ABB RobotStudio station: NLP2Commands_IRB140.rspag

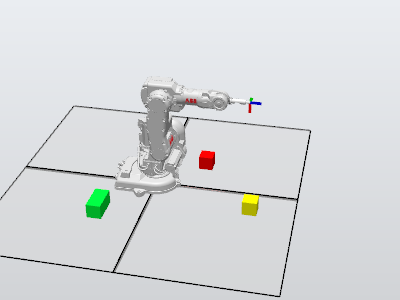
--- station ---
Station FinalProject (saved by RobotStudio 24.4.11080.0)
Controller IRB140_6_81
  mechanical unit ROB_1: IRB140_6_81, 6 joints, base frame (0, 0, 0) mm
Layout (positions relative to the parent item):
  - IRB140_6_81 [mechanism, from %ABB.RobotStudio.Models.IRB140%\IRB140_6_81_C_G_03.rslib] at (0, 0, 0) mm; joint values [0, 0, 0, 0, 0, 0] (rad or m)
  - VacuumGripper [mechanism] at (515, 0, 712) mm, rotated rx 0 ry 90 rz 0 deg
      TCP VacuumGripper at (122.78, 0, 0) mm, rotated rx 90 ry 45 rz 90 deg
      links: FakeEE
  - Cubo rojo [part] at (9, 9, 0) mm, size 100 x 100 x 100 mm
  - Cubo amarillo [part] at (0, 0, 0) mm, size 100 x 100 x 100 mm
  - Rectángulo verde [part] at (0, 0, 0) mm, size 100 x 200 x 100 mm
  - Cubo rojo [smart component, from Components\Positioner.rslib]
      properties: Object=Cubo rojo; Position=[0.009 0.009 0]; Orientation=[0 0 0]; Reference=Global; ReferenceObject=(none)
  - Cubo amarillo [smart component, from Components\Positioner.rslib]
      properties: Object=Cubo amarillo; Position=[0 0 0]; Orientation=[0 0 0]; Reference=Global; ReferenceObject=(none)
  - Rectángulo verde [smart component, from Components\Positioner.rslib]
      properties: Object=Rectángulo verde; Position=[0 0 0]; Orientation=[0 0 0]; Reference=Global; ReferenceObject=(none)
  - Detacher [smart component, from Components\Detacher.rslib]
      properties: Child=Cubo rojo; KeepPosition=true
  - Detacher_2 [smart component, from Components\Detacher.rslib]
      properties: Child=Cubo amarillo; KeepPosition=true
  - Detacher_3 [smart component, from Components\Detacher.rslib]
      properties: Child=Rectángulo verde; KeepPosition=true
  - Attacher [smart component, from Components\Attacher.rslib]
      properties: Parent=VacuumGripper; Flange=0; Child=Cubo rojo; Mount=false; Offset=[0 0 0]; Orientation=[0 0 0]
  - Attacher_2 [smart component, from Components\Attacher.rslib]
      properties: Parent=VacuumGripper; Flange=0; Child=Cubo amarillo; Mount=false; Offset=[0 0 0]; Orientation=[0 0 0]
  - Attacher_3 [smart component, from Components\Attacher.rslib]
      properties: Parent=VacuumGripper; Flange=0; Child=Rectángulo verde; Mount=false; Offset=[0 0 0]; Orientation=[0 0 0]
  - PlaneSensor [smart component, from Components\PlaneSensor.rslib]
      properties: Origin=[0.25 0.25 0.101]; Axis1=[0.1 0 0]; Axis2=[0 0.1 0]; Tag=(none); SensedPart=(none)
    - _sensorPart_ [part], size 100 x 100 x 0 mm
  - PlaneSensor_2 [smart component, from Components\PlaneSensor.rslib]
      properties: Origin=[0.65 -0.25 0.101]; Axis1=[0.1 0 0]; Axis2=[0 0.1 0]; Tag=(none); SensedPart=Cubo amarillo
    - _sensorPart_ [part], size 100 x 100 x 0 mm
  - PlaneSensor_3 [smart component, from Components\PlaneSensor.rslib]
      properties: Origin=[-0.35 -0.5 0.101]; Axis1=[0.1 0 0]; Axis2=[0 0.2 0]; Tag=(none); SensedPart=(none)
    - _sensorPart_ [part], size 100 x 200 x 0 mm
Attachment: VacuumGripper is attached to IRB140_6_81 / Link6
Station signals: DI Reset_posiciones
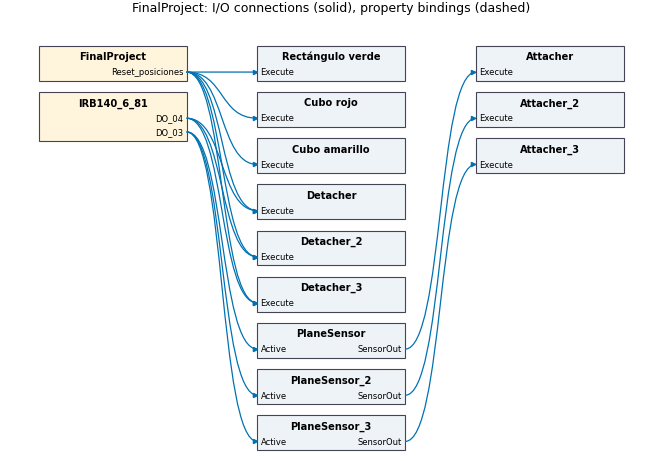
Station logic (signal -> signal, property => property):
  FinalProject.Reset_posiciones -> Rectángulo verde.Execute
  FinalProject.Reset_posiciones -> Cubo rojo.Execute
  FinalProject.Reset_posiciones -> Cubo amarillo.Execute
  IRB140_6_81.DO_04 -> Detacher.Execute
  IRB140_6_81.DO_04 -> Detacher_2.Execute
  IRB140_6_81.DO_04 -> Detacher_3.Execute
  FinalProject.Reset_posiciones -> Detacher.Execute
  FinalProject.Reset_posiciones -> Detacher_2.Execute
  FinalProject.Reset_posiciones -> Detacher_3.Execute
  PlaneSensor.SensorOut -> Attacher.Execute
  PlaneSensor_2.SensorOut -> Attacher_2.Execute
  PlaneSensor_3.SensorOut -> Attacher_3.Execute
  IRB140_6_81.DO_03 -> PlaneSensor.Active
  IRB140_6_81.DO_03 -> PlaneSensor_2.Active
  IRB140_6_81.DO_03 -> PlaneSensor_3.Active
Targets, tools, work objects and paths stored in the station and not in the controller backup, written as RAPID:
! task T_ROB1
MODULE Numbers
  CONST robtarget T_01:=[[-310.742,318.894,0],[1,0,0,0],[0,0,0,0],[9E+09,9E+09,9E+09,9E+09,9E+09,9E+09]];
  CONST robtarget T_02:=[[-285.702,367.273,0],[1,0,0,0],[0,-1,0,0],[9E+09,9E+09,9E+09,9E+09,9E+09,9E+09]];
  CONST robtarget T_03:=[[-206.529,382.913,0],[1,0,0,0],[0,-1,0,0],[9E+09,9E+09,9E+09,9E+09,9E+09,9E+09]];
  CONST robtarget T_04:=[[-128.165,367.435,0],[1,0,0,0],[0,-2,1,0],[9E+09,9E+09,9E+09,9E+09,9E+09,9E+09]];
  CONST robtarget T_05:=[[-102.477,318.894,0],[1,0,0,0],[-2,0,1,6],[9E+09,9E+09,9E+09,9E+09,9E+09,9E+09]];
  CONST robtarget T_06:=[[-127.679,270.676,0],[1,0,0,0],[-2,0,1,6],[9E+09,9E+09,9E+09,9E+09,9E+09,9E+09]];
  CONST robtarget T_07:=[[-206.691,255.036,0],[1,0,0,0],[-1,0,-1,0],[9E+09,9E+09,9E+09,9E+09,9E+09,9E+09]];
  CONST robtarget T_08:=[[-284.811,270.514,0],[1,0,0,0],[-1,0,-1,0],[9E+09,9E+09,9E+09,9E+09,9E+09,9E+09]];
  CONST robtarget T_09:=[[-310.742,318.894,0],[1,0,0,0],[0,-1,0,0],[9E+09,9E+09,9E+09,9E+09,9E+09,9E+09]];
  CONST robtarget T_11:=[[-106.691,366.707,0],[1,0,0,0],[0,0,-1,1],[9E+09,9E+09,9E+09,9E+09,9E+09,9E+09]];
  CONST robtarget T_12:=[[-106.691,269.138,0],[1,0,0,0],[0,0,-1,1],[9E+09,9E+09,9E+09,9E+09,9E+09,9E+09]];
  CONST robtarget T_13:=[[-106.691,317.923,0],[1,0,0,0],[0,0,-1,1],[9E+09,9E+09,9E+09,9E+09,9E+09,9E+09]];
  CONST robtarget T_14:=[[-307.339,315.005,0],[1,0,0,0],[0,0,-1,1],[9E+09,9E+09,9E+09,9E+09,9E+09,9E+09]];
  CONST robtarget T_15:=[[-285.297,336.399,0],[1,0,0,0],[0,1,-2,1],[9E+09,9E+09,9E+09,9E+09,9E+09,9E+09]];
  CONST robtarget T_16:=[[-279.462,366.707,0],[1,0,0,0],[0,1,-2,1],[9E+09,9E+09,9E+09,9E+09,9E+09,9E+09]];
  CONST robtarget T_21:=[[-106.691,261.009,0],[1,0,0,0],[0,-1,0,0],[9E+09,9E+09,9E+09,9E+09,9E+09,9E+09]];
  CONST robtarget T_22:=[[-106.691,384.347,0],[1,0,0,0],[0,-2,1,0],[9E+09,9E+09,9E+09,9E+09,9E+09,9E+09]];
  CONST robtarget T_23:=[[-129.867,359.226,0],[1,0,0,0],[0,-2,1,0],[9E+09,9E+09,9E+09,9E+09,9E+09,9E+09]];
  CONST robtarget T_24:=[[-153.206,334.509,0],[1,0,0,0],[0,-2,1,0],[9E+09,9E+09,9E+09,9E+09,9E+09,9E+09]];
  CONST robtarget T_25:=[[-181.731,306.39,0],[1,0,0,0],[0,-1,0,0],[9E+09,9E+09,9E+09,9E+09,9E+09,9E+09]];
  CONST robtarget T_26:=[[-215.929,279.647,0],[1,0,0,0],[0,-1,0,0],[9E+09,9E+09,9E+09,9E+09,9E+09,9E+09]];
  CONST robtarget T_27:=[[-255.961,269.274,0],[1,0,0,0],[0,-1,0,0],[9E+09,9E+09,9E+09,9E+09,9E+09,9E+09]];
  CONST robtarget T_28:=[[-296.075,285.077,0],[1,0,0,0],[0,-1,0,0],[9E+09,9E+09,9E+09,9E+09,9E+09,9E+09]];
  CONST robtarget T_29:=[[-310.905,328.918,0],[1,0,0,0],[0,-1,0,0],[9E+09,9E+09,9E+09,9E+09,9E+09,9E+09]];
  CONST robtarget T_210:=[[-306.934,357.038,0],[1,0,0,0],[0,-1,0,0],[9E+09,9E+09,9E+09,9E+09,9E+09,9E+09]];
  CONST robtarget T_211:=[[-298.911,380.133,0],[1,0,0,0],[0,-1,0,0],[9E+09,9E+09,9E+09,9E+09,9E+09,9E+09]];
  CONST robtarget T_31:=[[-298.587,375.377,0],[1,0,0,0],[0,-1,0,0],[9E+09,9E+09,9E+09,9E+09,9E+09,9E+09]];
  CONST robtarget T_32:=[[-307.096,351.633,0],[1,0,0,0],[0,-1,0,0],[9E+09,9E+09,9E+09,9E+09,9E+09,9E+09]];
  CONST robtarget T_33:=[[-310.905,323.189,0],[1,0,0,0],[0,-1,0,0],[9E+09,9E+09,9E+09,9E+09,9E+09,9E+09]];
  CONST robtarget T_34:=[[-308.149,299.445,0],[1,0,0,0],[0,-1,0,0],[9E+09,9E+09,9E+09,9E+09,9E+09,9E+09]];
  CONST robtarget T_35:=[[-299.559,281.049,0],[1,0,0,0],[0,-1,0,0],[9E+09,9E+09,9E+09,9E+09,9E+09,9E+09]];
  CONST robtarget T_36:=[[-284.081,267.759,0],[1,0,0,0],[0,-1,0,0],[9E+09,9E+09,9E+09,9E+09,9E+09,9E+09]];
  CONST robtarget T_37:=[[-262.606,263.221,0],[1,0,0,0],[0,-1,0,0],[9E+09,9E+09,9E+09,9E+09,9E+09,9E+09]];
  CONST robtarget T_38:=[[-233.595,274.08,0],[1,0,0,0],[0,-1,0,0],[9E+09,9E+09,9E+09,9E+09,9E+09,9E+09]];
  CONST robtarget T_39:=[[-217.874,300.174,0],[1,0,0,0],[0,-1,0,0],[9E+09,9E+09,9E+09,9E+09,9E+09,9E+09]];
  CONST robtarget T_310:=[[-215.199,340.044,0],[1,0,0,0],[0,-1,0,0],[9E+09,9E+09,9E+09,9E+09,9E+09,9E+09]];
  CONST robtarget T_311:=[[-215.929,300.174,0],[1,0,0,0],[0,-1,0,0],[9E+09,9E+09,9E+09,9E+09,9E+09,9E+09]];
  CONST robtarget T_312:=[[-202.963,273.27,0],[1,0,0,0],[0,-1,0,0],[9E+09,9E+09,9E+09,9E+09,9E+09,9E+09]];
  CONST robtarget T_313:=[[-188.214,263.221,0],[1,0,0,0],[0,-1,0,0],[9E+09,9E+09,9E+09,9E+09,9E+09,9E+09]];
  CONST robtarget T_314:=[[-166.01,259.331,0],[1,0,0,0],[0,-1,0,0],[9E+09,9E+09,9E+09,9E+09,9E+09,9E+09]];
  CONST robtarget T_315:=[[-141.131,263.95,0],[1,0,0,0],[0,-1,0,0],[9E+09,9E+09,9E+09,9E+09,9E+09,9E+09]];
  CONST robtarget T_316:=[[-120.953,276.997,0],[1,0,0,0],[0,-1,0,0],[9E+09,9E+09,9E+09,9E+09,9E+09,9E+09]];
  CONST robtarget T_317:=[[-107.177,298.148,0],[1,0,0,0],[0,-2,1,0],[9E+09,9E+09,9E+09,9E+09,9E+09,9E+09]];
  CONST robtarget T_318:=[[-102.477,326.268,0],[1,0,0,0],[0,-2,1,0],[9E+09,9E+09,9E+09,9E+09,9E+09,9E+09]];
  CONST robtarget T_319:=[[-106.123,356.09,0],[1,0,0,0],[0,-2,1,0],[9E+09,9E+09,9E+09,9E+09,9E+09,9E+09]];
  CONST robtarget T_320:=[[-114.794,380.887,0],[1,0,0,0],[0,-2,1,0],[9E+09,9E+09,9E+09,9E+09,9E+09,9E+09]];
  CONST robtarget T_41:=[[-106.691,281.323,0],[1,0,0,0],[-1,-1,0,1],[9E+09,9E+09,9E+09,9E+09,9E+09,9E+09]];
  CONST robtarget T_42:=[[-306.691,281.323,0],[1,0,0,0],[0,0,-1,1],[9E+09,9E+09,9E+09,9E+09,9E+09,9E+09]];
  CONST robtarget T_43:=[[-306.691,305.958,0],[1,0,0,0],[0,1,-2,1],[9E+09,9E+09,9E+09,9E+09,9E+09,9E+09]];
  CONST robtarget T_44:=[[-203.611,395.424,0],[1,0,0,0],[0,1,-2,1],[9E+09,9E+09,9E+09,9E+09,9E+09,9E+09]];
  CONST robtarget T_45:=[[-175.41,395.424,0],[1,0,0,0],[0,1,-2,1],[9E+09,9E+09,9E+09,9E+09,9E+09,9E+09]];
  CONST robtarget T_46:=[[-175.41,257.498,0],[1,0,0,0],[0,1,-2,1],[9E+09,9E+09,9E+09,9E+09,9E+09,9E+09]];
  CONST robtarget T_51:=[[-306.691,269.007,0],[1,0,0,0],[0,1,-2,1],[9E+09,9E+09,9E+09,9E+09,9E+09,9E+09]];
  CONST robtarget T_52:=[[-306.691,378.732,0],[1,0,0,0],[0,1,-2,1],[9E+09,9E+09,9E+09,9E+09,9E+09,9E+09]];
  CONST robtarget T_53:=[[-223.611,378.732,0],[1,0,0,0],[0,1,-2,1],[9E+09,9E+09,9E+09,9E+09,9E+09,9E+09]];
  CONST robtarget T_54:=[[-229.867,352.962,0],[1,0,0,0],[0,1,-2,1],[9E+09,9E+09,9E+09,9E+09,9E+09,9E+09]];
  CONST robtarget T_55:=[[-231.002,334.809,0],[1,0,0,0],[0,1,-2,1],[9E+09,9E+09,9E+09,9E+09,9E+09,9E+09]];
  CONST robtarget T_56:=[[-228.49,308.796,0],[1,0,0,0],[0,1,-2,1],[9E+09,9E+09,9E+09,9E+09,9E+09,9E+09]];
  CONST robtarget T_57:=[[-218.522,288.456,0],[1,0,0,0],[0,1,-2,1],[9E+09,9E+09,9E+09,9E+09,9E+09,9E+09]];
  CONST robtarget T_58:=[[-199.721,273.221,0],[1,0,0,0],[0,1,-2,1],[9E+09,9E+09,9E+09,9E+09,9E+09,9E+09]];
  CONST robtarget T_59:=[[-170.224,267.873,0],[1,0,0,0],[0,1,-2,1],[9E+09,9E+09,9E+09,9E+09,9E+09,9E+09]];
  CONST robtarget T_510:=[[-143.482,272.492,0],[1,0,0,0],[0,0,-1,1],[9E+09,9E+09,9E+09,9E+09,9E+09,9E+09]];
  CONST robtarget T_511:=[[-122.088,285.539,0],[1,0,0,0],[0,0,-1,1],[9E+09,9E+09,9E+09,9E+09,9E+09,9E+09]];
  CONST robtarget T_512:=[[-107.744,306.527,0],[1,0,0,0],[0,0,-1,1],[9E+09,9E+09,9E+09,9E+09,9E+09,9E+09]];
  CONST robtarget T_513:=[[-102.477,334.647,0],[1,0,0,0],[0,0,-1,1],[9E+09,9E+09,9E+09,9E+09,9E+09,9E+09]];
  CONST robtarget T_514:=[[-105.637,362.848,0],[1,0,0,0],[0,0,-1,1],[9E+09,9E+09,9E+09,9E+09,9E+09,9E+09]];
  CONST robtarget T_515:=[[-113.822,386.997,0],[1,0,0,0],[0,0,-1,1],[9E+09,9E+09,9E+09,9E+09,9E+09,9E+09]];
  CONST robtarget T_61:=[[-307.663,280.947,0],[1,0,0,0],[0,0,-1,1],[9E+09,9E+09,9E+09,9E+09,9E+09,9E+09]];
  CONST robtarget T_62:=[[-310.418,303.638,0],[1,0,0,0],[0,1,-2,1],[9E+09,9E+09,9E+09,9E+09,9E+09,9E+09]];
  CONST robtarget T_63:=[[-301.909,343.346,0],[1,0,0,0],[0,1,-2,1],[9E+09,9E+09,9E+09,9E+09,9E+09,9E+09]];
  CONST robtarget T_64:=[[-278.165,371.385,0],[1,0,0,0],[0,1,-2,1],[9E+09,9E+09,9E+09,9E+09,9E+09,9E+09]];
  CONST robtarget T_65:=[[-241.618,387.916,0],[1,0,0,0],[0,1,-2,1],[9E+09,9E+09,9E+09,9E+09,9E+09,9E+09]];
  CONST robtarget T_66:=[[-194.535,393.265,0],[1,0,0,0],[0,1,-2,1],[9E+09,9E+09,9E+09,9E+09,9E+09,9E+09]];
  CONST robtarget T_67:=[[-149.721,387.43,0],[1,0,0,0],[0,1,-2,1],[9E+09,9E+09,9E+09,9E+09,9E+09,9E+09]];
  CONST robtarget T_68:=[[-120.629,371.223,0],[1,0,0,0],[0,0,-1,1],[9E+09,9E+09,9E+09,9E+09,9E+09,9E+09]];
  CONST robtarget T_69:=[[-107.015,351.693,0],[1,0,0,0],[0,0,-1,1],[9E+09,9E+09,9E+09,9E+09,9E+09,9E+09]];
  CONST robtarget T_610:=[[-102.477,327.138,0],[1,0,0,0],[0,0,-1,1],[9E+09,9E+09,9E+09,9E+09,9E+09,9E+09]];
  CONST robtarget T_611:=[[-107.258,302.503,0],[1,0,0,0],[0,0,-1,1],[9E+09,9E+09,9E+09,9E+09,9E+09,9E+09]];
  CONST robtarget T_612:=[[-121.277,282.406,0],[1,0,0,0],[0,0,-1,1],[9E+09,9E+09,9E+09,9E+09,9E+09,9E+09]];
  CONST robtarget T_613:=[[-143.076,268.71,0],[1,0,0,0],[0,0,-1,1],[9E+09,9E+09,9E+09,9E+09,9E+09,9E+09]];
  CONST robtarget T_614:=[[-171.52,263.605,0],[1,0,0,0],[0,1,-2,1],[9E+09,9E+09,9E+09,9E+09,9E+09,9E+09]];
  CONST robtarget T_615:=[[-201.504,268.954,0],[1,0,0,0],[0,1,-2,1],[9E+09,9E+09,9E+09,9E+09,9E+09,9E+09]];
  CONST robtarget T_616:=[[-222.574,285.323,0],[1,0,0,0],[0,1,-2,1],[9E+09,9E+09,9E+09,9E+09,9E+09,9E+09]];
  CONST robtarget T_617:=[[-232.055,303.638,0],[1,0,0,0],[0,1,-2,1],[9E+09,9E+09,9E+09,9E+09,9E+09,9E+09]];
  CONST robtarget T_618:=[[-234.405,324.059,0],[1,0,0,0],[0,1,-2,1],[9E+09,9E+09,9E+09,9E+09,9E+09,9E+09]];
  CONST robtarget T_619:=[[-230.759,346.101,0],[1,0,0,0],[0,1,-2,1],[9E+09,9E+09,9E+09,9E+09,9E+09,9E+09]];
  CONST robtarget T_620:=[[-220.467,365.712,0],[1,0,0,0],[0,1,-2,1],[9E+09,9E+09,9E+09,9E+09,9E+09,9E+09]];
  CONST robtarget T_621:=[[-194.535,393.265,0],[1,0,0,0],[0,1,-2,1],[9E+09,9E+09,9E+09,9E+09,9E+09,9E+09]];
  CONST robtarget T_71:=[[-306.691,388.239,0],[1,0,0,0],[0,-1,0,0],[9E+09,9E+09,9E+09,9E+09,9E+09,9E+09]];
  CONST robtarget T_72:=[[-306.691,261.334,0],[1,0,0,0],[0,-1,0,0],[9E+09,9E+09,9E+09,9E+09,9E+09,9E+09]];
  CONST robtarget T_73:=[[-106.691,347.882,0],[1,0,0,0],[0,-1,0,0],[9E+09,9E+09,9E+09,9E+09,9E+09,9E+09]];
  CONST robtarget T_81:=[[-214.308,359.688,0],[1,0,0,0],[0,1,-2,1],[9E+09,9E+09,9E+09,9E+09,9E+09,9E+09]];
  CONST robtarget T_82:=[[-233.109,381.568,0],[1,0,0,0],[0,1,-2,1],[9E+09,9E+09,9E+09,9E+09,9E+09,9E+09]];
  CONST robtarget T_83:=[[-258.554,388.699,0],[1,0,0,0],[0,1,-2,1],[9E+09,9E+09,9E+09,9E+09,9E+09,9E+09]];
  CONST robtarget T_84:=[[-296.156,371.681,0],[1,0,0,0],[0,1,-2,1],[9E+09,9E+09,9E+09,9E+09,9E+09,9E+09]];
  CONST robtarget T_85:=[[-311.229,328.407,0],[1,0,0,0],[0,1,-2,1],[9E+09,9E+09,9E+09,9E+09,9E+09,9E+09]];
  CONST robtarget T_86:=[[-296.966,284.728,0],[1,0,0,0],[0,1,-2,1],[9E+09,9E+09,9E+09,9E+09,9E+09,9E+09]];
  CONST robtarget T_87:=[[-260.337,268.278,0],[1,0,0,0],[0,1,-2,1],[9E+09,9E+09,9E+09,9E+09,9E+09,9E+09]];
  CONST robtarget T_88:=[[-233.757,276.138,0],[1,0,0,0],[0,1,-2,1],[9E+09,9E+09,9E+09,9E+09,9E+09,9E+09]];
  CONST robtarget T_89:=[[-213.174,298.748,0],[1,0,0,0],[0,1,-2,1],[9E+09,9E+09,9E+09,9E+09,9E+09,9E+09]];
  CONST robtarget T_810:=[[-213.498,359.688,0],[1,0,0,0],[0,1,-2,1],[9E+09,9E+09,9E+09,9E+09,9E+09,9E+09]];
  CONST robtarget T_811:=[[-191.78,384.89,0],[1,0,0,0],[0,1,-2,1],[9E+09,9E+09,9E+09,9E+09,9E+09,9E+09]];
  CONST robtarget T_812:=[[-161.958,393.561,0],[1,0,0,0],[0,1,-2,1],[9E+09,9E+09,9E+09,9E+09,9E+09,9E+09]];
  CONST robtarget T_813:=[[-138.457,389.185,0],[1,0,0,0],[0,0,-1,1],[9E+09,9E+09,9E+09,9E+09,9E+09,9E+09]];
  CONST robtarget T_814:=[[-119.332,376.381,0],[1,0,0,0],[0,0,-1,1],[9E+09,9E+09,9E+09,9E+09,9E+09,9E+09]];
  CONST robtarget T_815:=[[-106.61,355.555,0],[1,0,0,0],[0,0,-1,1],[9E+09,9E+09,9E+09,9E+09,9E+09,9E+09]];
  CONST robtarget T_816:=[[-102.152,328.407,0],[1,0,0,0],[0,0,-1,1],[9E+09,9E+09,9E+09,9E+09,9E+09,9E+09]];
  CONST robtarget T_817:=[[-119.494,281.892,0],[1,0,0,0],[0,0,-1,1],[9E+09,9E+09,9E+09,9E+09,9E+09,9E+09]];
  CONST robtarget T_818:=[[-162.444,263.253,0],[1,0,0,0],[0,1,-2,1],[9E+09,9E+09,9E+09,9E+09,9E+09,9E+09]];
  CONST robtarget T_819:=[[-192.59,272.249,0],[1,0,0,0],[0,1,-2,1],[9E+09,9E+09,9E+09,9E+09,9E+09,9E+09]];
  CONST robtarget T_820:=[[-212.363,298.748,0],[1,0,0,0],[0,1,-2,1],[9E+09,9E+09,9E+09,9E+09,9E+09,9E+09]];
  CONST robtarget T_821:=[[-214.308,359.688,0],[1,0,0,0],[0,1,-2,1],[9E+09,9E+09,9E+09,9E+09,9E+09,9E+09]];
  CONST robtarget T_91:=[[-105.556,371.949,0],[1,0,0,0],[0,0,-1,1],[9E+09,9E+09,9E+09,9E+09,9E+09,9E+09]];
  CONST robtarget T_92:=[[-102.801,349.258,0],[1,0,0,0],[0,0,-1,1],[9E+09,9E+09,9E+09,9E+09,9E+09,9E+09]];
  CONST robtarget T_93:=[[-110.986,309.388,0],[1,0,0,0],[0,0,-1,1],[9E+09,9E+09,9E+09,9E+09,9E+09,9E+09]];
  CONST robtarget T_94:=[[-134.729,281.673,0],[1,0,0,0],[0,0,-1,1],[9E+09,9E+09,9E+09,9E+09,9E+09,9E+09]];
  CONST robtarget T_95:=[[-171.682,265.223,0],[1,0,0,0],[0,1,-2,1],[9E+09,9E+09,9E+09,9E+09,9E+09,9E+09]];
  CONST robtarget T_96:=[[-218.684,259.631,0],[1,0,0,0],[0,1,-2,1],[9E+09,9E+09,9E+09,9E+09,9E+09,9E+09]];
  CONST robtarget T_97:=[[-263.903,265.304,0],[1,0,0,0],[0,1,-2,1],[9E+09,9E+09,9E+09,9E+09,9E+09,9E+09]];
  CONST robtarget T_98:=[[-292.752,281.349,0],[1,0,0,0],[0,1,-2,1],[9E+09,9E+09,9E+09,9E+09,9E+09,9E+09]];
  CONST robtarget T_99:=[[-306.123,300.798,0],[1,0,0,0],[0,1,-2,1],[9E+09,9E+09,9E+09,9E+09,9E+09,9E+09]];
  CONST robtarget T_910:=[[-310.742,325.757,0],[1,0,0,0],[0,1,-2,1],[9E+09,9E+09,9E+09,9E+09,9E+09,9E+09]];
  CONST robtarget T_911:=[[-305.799,350.15,0],[1,0,0,0],[0,1,-2,1],[9E+09,9E+09,9E+09,9E+09,9E+09,9E+09]];
  CONST robtarget T_912:=[[-291.942,370.49,0],[1,0,0,0],[0,1,-2,1],[9E+09,9E+09,9E+09,9E+09,9E+09,9E+09]];
  CONST robtarget T_913:=[[-269.9,384.266,0],[1,0,0,0],[0,1,-2,1],[9E+09,9E+09,9E+09,9E+09,9E+09,9E+09]];
  CONST robtarget T_914:=[[-241.699,389.291,0],[1,0,0,0],[0,1,-2,1],[9E+09,9E+09,9E+09,9E+09,9E+09,9E+09]];
  CONST robtarget T_915:=[[-211.472,383.78,0],[1,0,0,0],[0,1,-2,1],[9E+09,9E+09,9E+09,9E+09,9E+09,9E+09]];
  CONST robtarget T_916:=[[-190.645,367.573,0],[1,0,0,0],[0,1,-2,1],[9E+09,9E+09,9E+09,9E+09,9E+09,9E+09]];
  CONST robtarget T_917:=[[-181.245,349.177,0],[1,0,0,0],[0,1,-2,1],[9E+09,9E+09,9E+09,9E+09,9E+09,9E+09]];
  CONST robtarget T_918:=[[-178.814,328.999,0],[1,0,0,0],[0,1,-2,1],[9E+09,9E+09,9E+09,9E+09,9E+09,9E+09]];
  CONST robtarget T_919:=[[-182.136,307.767,0],[1,0,0,0],[0,1,-2,1],[9E+09,9E+09,9E+09,9E+09,9E+09,9E+09]];
  CONST robtarget T_920:=[[-192.752,287.346,0],[1,0,0,0],[0,1,-2,1],[9E+09,9E+09,9E+09,9E+09,9E+09,9E+09]];
  CONST robtarget T_921:=[[-218.684,259.631,0],[1,0,0,0],[0,1,-2,1],[9E+09,9E+09,9E+09,9E+09,9E+09,9E+09]];
  CONST robtarget T_921_2:=[[-218.684,259.631,0],[1,0,0,0],[-1,-2,1,1],[9E+09,9E+09,9E+09,9E+09,9E+09,9E+09]];
  CONST robtarget T_01_2:=[[-310.742,318.894,0],[1,0,0,0],[0,0,0,0],[9E+09,9E+09,9E+09,9E+09,9E+09,9E+09]];
  CONST robtarget T_02_2:=[[-285.702,367.273,0],[1,0,0,0],[-1,0,-1,0],[9E+09,9E+09,9E+09,9E+09,9E+09,9E+09]];
  CONST robtarget T_03_2:=[[-206.529,382.913,0],[1,0,0,0],[-1,0,-1,0],[9E+09,9E+09,9E+09,9E+09,9E+09,9E+09]];
  CONST robtarget T_04_2:=[[-128.165,367.435,0],[1,0,0,0],[-1,0,-1,0],[9E+09,9E+09,9E+09,9E+09,9E+09,9E+09]];
  CONST robtarget T_05_2:=[[-102.477,318.894,0],[1,0,0,0],[-1,0,-1,0],[9E+09,9E+09,9E+09,9E+09,9E+09,9E+09]];
  CONST robtarget T_06_2:=[[-127.679,270.676,0],[1,0,0,0],[-1,1,-2,0],[9E+09,9E+09,9E+09,9E+09,9E+09,9E+09]];
  CONST robtarget T_07_2:=[[-206.691,255.036,0],[1,0,0,0],[-1,0,-1,0],[9E+09,9E+09,9E+09,9E+09,9E+09,9E+09]];
  CONST robtarget T_08_2:=[[-284.811,270.514,0],[1,0,0,0],[-1,0,-1,0],[9E+09,9E+09,9E+09,9E+09,9E+09,9E+09]];
  CONST robtarget T_09_2:=[[-310.742,318.894,0],[1,0,0,0],[-1,0,-1,0],[9E+09,9E+09,9E+09,9E+09,9E+09,9E+09]];
  CONST robtarget T_11_2:=[[-106.691,366.707,0],[1,0,0,0],[-1,1,-2,0],[9E+09,9E+09,9E+09,9E+09,9E+09,9E+09]];
  CONST robtarget T_12_2:=[[-106.691,269.138,0],[1,0,0,0],[-1,1,-2,0],[9E+09,9E+09,9E+09,9E+09,9E+09,9E+09]];
  CONST robtarget T_13_2:=[[-106.691,317.923,0],[1,0,0,0],[-1,1,-2,0],[9E+09,9E+09,9E+09,9E+09,9E+09,9E+09]];
  CONST robtarget T_14_2:=[[-307.339,315.005,0],[1,0,0,0],[-1,1,-2,0],[9E+09,9E+09,9E+09,9E+09,9E+09,9E+09]];
  CONST robtarget T_15_2:=[[-285.297,336.399,0],[1,0,0,0],[-1,0,-1,0],[9E+09,9E+09,9E+09,9E+09,9E+09,9E+09]];
  CONST robtarget T_16_2:=[[-279.462,366.707,0],[1,0,0,0],[-1,0,-1,0],[9E+09,9E+09,9E+09,9E+09,9E+09,9E+09]];
  CONST robtarget T_21_2:=[[-106.691,261.009,0],[1,0,0,0],[-1,1,-2,0],[9E+09,9E+09,9E+09,9E+09,9E+09,9E+09]];
  CONST robtarget T_22_2:=[[-106.691,384.347,0],[1,0,0,0],[-1,1,-2,0],[9E+09,9E+09,9E+09,9E+09,9E+09,9E+09]];
  CONST robtarget T_23_2:=[[-129.867,359.226,0],[1,0,0,0],[-1,1,-2,0],[9E+09,9E+09,9E+09,9E+09,9E+09,9E+09]];
  CONST robtarget T_24_2:=[[-153.206,334.509,0],[1,0,0,0],[-1,0,-1,0],[9E+09,9E+09,9E+09,9E+09,9E+09,9E+09]];
  CONST robtarget T_25_2:=[[-181.731,306.39,0],[1,0,0,0],[-1,0,-1,0],[9E+09,9E+09,9E+09,9E+09,9E+09,9E+09]];
  CONST robtarget T_26_2:=[[-215.929,279.647,0],[1,0,0,0],[-1,0,-1,0],[9E+09,9E+09,9E+09,9E+09,9E+09,9E+09]];
  CONST robtarget T_27_2:=[[-255.961,269.274,0],[1,0,0,0],[-1,0,-1,0],[9E+09,9E+09,9E+09,9E+09,9E+09,9E+09]];
  CONST robtarget T_28_2:=[[-296.075,285.077,0],[1,0,0,0],[-1,0,-1,0],[9E+09,9E+09,9E+09,9E+09,9E+09,9E+09]];
  CONST robtarget T_29_2:=[[-310.905,328.918,0],[1,0,0,0],[-1,0,-1,0],[9E+09,9E+09,9E+09,9E+09,9E+09,9E+09]];
  CONST robtarget T_210_2:=[[-306.934,357.038,0],[1,0,0,0],[-1,0,-1,0],[9E+09,9E+09,9E+09,9E+09,9E+09,9E+09]];
  CONST robtarget T_211_2:=[[-298.911,380.133,0],[1,0,0,0],[-1,0,-1,0],[9E+09,9E+09,9E+09,9E+09,9E+09,9E+09]];
  CONST robtarget T_31_2:=[[-298.587,375.377,0],[1,0,0,0],[0,-1,0,0],[9E+09,9E+09,9E+09,9E+09,9E+09,9E+09]];
  CONST robtarget T_32_2:=[[-307.096,351.633,0],[1,0,0,0],[-1,0,-1,0],[9E+09,9E+09,9E+09,9E+09,9E+09,9E+09]];
  CONST robtarget T_33_2:=[[-310.905,323.189,0],[1,0,0,0],[-1,0,-1,0],[9E+09,9E+09,9E+09,9E+09,9E+09,9E+09]];
  CONST robtarget T_34_2:=[[-308.149,299.445,0],[1,0,0,0],[-1,0,-1,0],[9E+09,9E+09,9E+09,9E+09,9E+09,9E+09]];
  CONST robtarget T_35_2:=[[-299.559,281.049,0],[1,0,0,0],[-1,0,-1,0],[9E+09,9E+09,9E+09,9E+09,9E+09,9E+09]];
  CONST robtarget T_36_2:=[[-284.081,267.759,0],[1,0,0,0],[-1,0,-1,0],[9E+09,9E+09,9E+09,9E+09,9E+09,9E+09]];
  CONST robtarget T_37_2:=[[-262.606,263.221,0],[1,0,0,0],[-1,0,-1,0],[9E+09,9E+09,9E+09,9E+09,9E+09,9E+09]];
  CONST robtarget T_38_2:=[[-233.595,274.08,0],[1,0,0,0],[-1,0,-1,0],[9E+09,9E+09,9E+09,9E+09,9E+09,9E+09]];
  CONST robtarget T_39_2:=[[-217.874,300.174,0],[1,0,0,0],[-1,0,-1,0],[9E+09,9E+09,9E+09,9E+09,9E+09,9E+09]];
  CONST robtarget T_310_2:=[[-215.199,340.044,0],[1,0,0,0],[0,-1,0,0],[9E+09,9E+09,9E+09,9E+09,9E+09,9E+09]];
  CONST robtarget T_311_2:=[[-215.929,300.174,0],[1,0,0,0],[0,-1,0,0],[9E+09,9E+09,9E+09,9E+09,9E+09,9E+09]];
  CONST robtarget T_312_2:=[[-202.963,273.27,0],[1,0,0,0],[0,-1,0,0],[9E+09,9E+09,9E+09,9E+09,9E+09,9E+09]];
  CONST robtarget T_313_2:=[[-188.214,263.221,0],[1,0,0,0],[0,-1,0,0],[9E+09,9E+09,9E+09,9E+09,9E+09,9E+09]];
  CONST robtarget T_314_2:=[[-166.01,259.331,0],[1,0,0,0],[0,-1,0,0],[9E+09,9E+09,9E+09,9E+09,9E+09,9E+09]];
  CONST robtarget T_315_2:=[[-141.131,263.95,0],[1,0,0,0],[0,-1,0,0],[9E+09,9E+09,9E+09,9E+09,9E+09,9E+09]];
  CONST robtarget T_316_2:=[[-120.953,276.997,0],[1,0,0,0],[-1,1,-2,0],[9E+09,9E+09,9E+09,9E+09,9E+09,9E+09]];
  CONST robtarget T_317_2:=[[-107.177,298.148,0],[1,0,0,0],[-1,1,-2,0],[9E+09,9E+09,9E+09,9E+09,9E+09,9E+09]];
  CONST robtarget T_318_2:=[[-102.477,326.268,0],[1,0,0,0],[-1,1,-2,0],[9E+09,9E+09,9E+09,9E+09,9E+09,9E+09]];
  CONST robtarget T_319_2:=[[-106.123,356.09,0],[1,0,0,0],[-1,1,-2,0],[9E+09,9E+09,9E+09,9E+09,9E+09,9E+09]];
  CONST robtarget T_320_2:=[[-114.794,380.887,0],[1,0,0,0],[0,-2,1,0],[9E+09,9E+09,9E+09,9E+09,9E+09,9E+09]];
  CONST robtarget T_41_2:=[[-106.691,281.323,0],[1,0,0,0],[-1,1,-2,0],[9E+09,9E+09,9E+09,9E+09,9E+09,9E+09]];
  CONST robtarget T_42_2:=[[-306.691,281.323,0],[1,0,0,0],[-1,0,-1,0],[9E+09,9E+09,9E+09,9E+09,9E+09,9E+09]];
  CONST robtarget T_43_2:=[[-306.691,305.958,0],[1,0,0,0],[-1,0,-1,0],[9E+09,9E+09,9E+09,9E+09,9E+09,9E+09]];
  CONST robtarget T_44_2:=[[-203.611,395.424,0],[1,0,0,0],[0,-1,0,0],[9E+09,9E+09,9E+09,9E+09,9E+09,9E+09]];
  CONST robtarget T_45_2:=[[-175.41,395.424,0],[1,0,0,0],[0,-1,0,0],[9E+09,9E+09,9E+09,9E+09,9E+09,9E+09]];
  CONST robtarget T_46_2:=[[-175.41,257.498,0],[1,0,0,0],[-1,0,-1,0],[9E+09,9E+09,9E+09,9E+09,9E+09,9E+09]];
  CONST robtarget T_51_2:=[[-306.691,269.007,0],[1,0,0,0],[-1,0,-1,0],[9E+09,9E+09,9E+09,9E+09,9E+09,9E+09]];
  CONST robtarget T_52_2:=[[-306.691,378.732,0],[1,0,0,0],[0,-1,0,0],[9E+09,9E+09,9E+09,9E+09,9E+09,9E+09]];
  CONST robtarget T_53_2:=[[-223.611,378.732,0],[1,0,0,0],[0,-1,0,0],[9E+09,9E+09,9E+09,9E+09,9E+09,9E+09]];
  CONST robtarget T_54_2:=[[-229.867,352.962,0],[1,0,0,0],[-1,0,-1,0],[9E+09,9E+09,9E+09,9E+09,9E+09,9E+09]];
  CONST robtarget T_55_2:=[[-231.002,334.809,0],[1,0,0,0],[-1,0,-1,0],[9E+09,9E+09,9E+09,9E+09,9E+09,9E+09]];
  CONST robtarget T_56_2:=[[-228.49,308.796,0],[1,0,0,0],[-1,0,-1,0],[9E+09,9E+09,9E+09,9E+09,9E+09,9E+09]];
  CONST robtarget T_57_2:=[[-218.522,288.456,0],[1,0,0,0],[-1,0,-1,0],[9E+09,9E+09,9E+09,9E+09,9E+09,9E+09]];
  CONST robtarget T_58_2:=[[-199.721,273.221,0],[1,0,0,0],[-1,0,-1,0],[9E+09,9E+09,9E+09,9E+09,9E+09,9E+09]];
  CONST robtarget T_59_2:=[[-170.224,267.873,0],[1,0,0,0],[-1,0,-1,0],[9E+09,9E+09,9E+09,9E+09,9E+09,9E+09]];
  CONST robtarget T_510_2:=[[-143.482,272.492,0],[1,0,0,0],[-1,0,-1,0],[9E+09,9E+09,9E+09,9E+09,9E+09,9E+09]];
  CONST robtarget T_511_2:=[[-122.088,285.539,0],[1,0,0,0],[0,0,-1,1],[9E+09,9E+09,9E+09,9E+09,9E+09,9E+09]];
  CONST robtarget T_512_2:=[[-107.744,306.527,0],[1,0,0,0],[0,0,-1,1],[9E+09,9E+09,9E+09,9E+09,9E+09,9E+09]];
  CONST robtarget T_513_2:=[[-102.477,334.647,0],[1,0,0,0],[0,0,-1,1],[9E+09,9E+09,9E+09,9E+09,9E+09,9E+09]];
  CONST robtarget T_514_2:=[[-105.637,362.848,0],[1,0,0,0],[0,0,-1,1],[9E+09,9E+09,9E+09,9E+09,9E+09,9E+09]];
  CONST robtarget T_515_2:=[[-113.822,386.997,0],[1,0,0,0],[0,0,-1,1],[9E+09,9E+09,9E+09,9E+09,9E+09,9E+09]];
  CONST robtarget T_61_2:=[[-307.663,280.947,0],[1,0,0,0],[-1,0,-1,0],[9E+09,9E+09,9E+09,9E+09,9E+09,9E+09]];
  CONST robtarget T_62_2:=[[-310.418,303.638,0],[1,0,0,0],[-1,0,-1,0],[9E+09,9E+09,9E+09,9E+09,9E+09,9E+09]];
  CONST robtarget T_63_2:=[[-301.909,343.346,0],[1,0,0,0],[-1,0,-1,0],[9E+09,9E+09,9E+09,9E+09,9E+09,9E+09]];
  CONST robtarget T_64_2:=[[-278.165,371.385,0],[1,0,0,0],[0,-1,0,0],[9E+09,9E+09,9E+09,9E+09,9E+09,9E+09]];
  CONST robtarget T_65_2:=[[-241.618,387.916,0],[1,0,0,0],[0,-1,0,0],[9E+09,9E+09,9E+09,9E+09,9E+09,9E+09]];
  CONST robtarget T_66_2:=[[-194.535,393.265,0],[1,0,0,0],[0,-1,0,0],[9E+09,9E+09,9E+09,9E+09,9E+09,9E+09]];
  CONST robtarget T_67_2:=[[-149.721,387.43,0],[1,0,0,0],[0,-1,0,0],[9E+09,9E+09,9E+09,9E+09,9E+09,9E+09]];
  CONST robtarget T_68_2:=[[-120.629,371.223,0],[1,0,0,0],[0,-1,0,0],[9E+09,9E+09,9E+09,9E+09,9E+09,9E+09]];
  CONST robtarget T_69_2:=[[-107.015,351.693,0],[1,0,0,0],[-1,1,-2,0],[9E+09,9E+09,9E+09,9E+09,9E+09,9E+09]];
  CONST robtarget T_610_2:=[[-102.477,327.138,0],[1,0,0,0],[0,0,-1,1],[9E+09,9E+09,9E+09,9E+09,9E+09,9E+09]];
  CONST robtarget T_611_2:=[[-107.258,302.503,0],[1,0,0,0],[0,0,-1,1],[9E+09,9E+09,9E+09,9E+09,9E+09,9E+09]];
  CONST robtarget T_612_2:=[[-121.277,282.406,0],[1,0,0,0],[0,0,-1,1],[9E+09,9E+09,9E+09,9E+09,9E+09,9E+09]];
  CONST robtarget T_613_2:=[[-143.076,268.71,0],[1,0,0,0],[-1,-2,1,1],[9E+09,9E+09,9E+09,9E+09,9E+09,9E+09]];
  CONST robtarget T_614_2:=[[-171.52,263.605,0],[1,0,0,0],[-1,-2,1,1],[9E+09,9E+09,9E+09,9E+09,9E+09,9E+09]];
  CONST robtarget T_615_2:=[[-201.504,268.954,0],[1,0,0,0],[-1,-2,1,1],[9E+09,9E+09,9E+09,9E+09,9E+09,9E+09]];
  CONST robtarget T_616_2:=[[-222.574,285.323,0],[1,0,0,0],[-1,-2,1,1],[9E+09,9E+09,9E+09,9E+09,9E+09,9E+09]];
  CONST robtarget T_617_2:=[[-232.055,303.638,0],[1,0,0,0],[-1,-2,1,1],[9E+09,9E+09,9E+09,9E+09,9E+09,9E+09]];
  CONST robtarget T_618_2:=[[-234.405,324.059,0],[1,0,0,0],[-1,-2,1,1],[9E+09,9E+09,9E+09,9E+09,9E+09,9E+09]];
  CONST robtarget T_619_2:=[[-230.759,346.101,0],[1,0,0,0],[-1,-2,1,1],[9E+09,9E+09,9E+09,9E+09,9E+09,9E+09]];
  CONST robtarget T_620_2:=[[-220.467,365.712,0],[1,0,0,0],[0,1,-2,1],[9E+09,9E+09,9E+09,9E+09,9E+09,9E+09]];
  CONST robtarget T_621_2:=[[-194.535,393.265,0],[1,0,0,0],[0,1,-2,1],[9E+09,9E+09,9E+09,9E+09,9E+09,9E+09]];
  CONST robtarget T_71_2:=[[-306.691,388.239,0],[1,0,0,0],[0,-1,0,0],[9E+09,9E+09,9E+09,9E+09,9E+09,9E+09]];
  CONST robtarget T_72_2:=[[-306.691,261.334,0],[1,0,0,0],[-1,0,-1,0],[9E+09,9E+09,9E+09,9E+09,9E+09,9E+09]];
  CONST robtarget T_73_2:=[[-106.691,347.882,0],[1,0,0,0],[-1,1,-2,0],[9E+09,9E+09,9E+09,9E+09,9E+09,9E+09]];
  CONST robtarget T_81_2:=[[-214.308,359.688,0],[1,0,0,0],[-1,0,-1,0],[9E+09,9E+09,9E+09,9E+09,9E+09,9E+09]];
  CONST robtarget T_82_2:=[[-233.109,381.568,0],[1,0,0,0],[0,-1,0,0],[9E+09,9E+09,9E+09,9E+09,9E+09,9E+09]];
  CONST robtarget T_83_2:=[[-258.554,388.699,0],[1,0,0,0],[0,-1,0,0],[9E+09,9E+09,9E+09,9E+09,9E+09,9E+09]];
  CONST robtarget T_84_2:=[[-296.156,371.681,0],[1,0,0,0],[0,-1,0,0],[9E+09,9E+09,9E+09,9E+09,9E+09,9E+09]];
  CONST robtarget T_85_2:=[[-311.229,328.407,0],[1,0,0,0],[-1,0,-1,0],[9E+09,9E+09,9E+09,9E+09,9E+09,9E+09]];
  CONST robtarget T_86_2:=[[-296.966,284.728,0],[1,0,0,0],[-1,0,-1,0],[9E+09,9E+09,9E+09,9E+09,9E+09,9E+09]];
  CONST robtarget T_87_2:=[[-260.337,268.278,0],[1,0,0,0],[-1,0,-1,0],[9E+09,9E+09,9E+09,9E+09,9E+09,9E+09]];
  CONST robtarget T_88_2:=[[-233.757,276.138,0],[1,0,0,0],[-1,0,-1,0],[9E+09,9E+09,9E+09,9E+09,9E+09,9E+09]];
  CONST robtarget T_89_2:=[[-213.174,298.748,0],[1,0,0,0],[-1,0,-1,0],[9E+09,9E+09,9E+09,9E+09,9E+09,9E+09]];
  CONST robtarget T_810_2:=[[-213.498,359.688,0],[1,0,0,0],[0,1,-2,1],[9E+09,9E+09,9E+09,9E+09,9E+09,9E+09]];
  CONST robtarget T_811_2:=[[-191.78,384.89,0],[1,0,0,0],[0,1,-2,1],[9E+09,9E+09,9E+09,9E+09,9E+09,9E+09]];
  CONST robtarget T_812_2:=[[-161.958,393.561,0],[1,0,0,0],[0,1,-2,1],[9E+09,9E+09,9E+09,9E+09,9E+09,9E+09]];
  CONST robtarget T_813_2:=[[-138.457,389.185,0],[1,0,0,0],[0,0,-1,1],[9E+09,9E+09,9E+09,9E+09,9E+09,9E+09]];
  CONST robtarget T_814_2:=[[-119.332,376.381,0],[1,0,0,0],[0,0,-1,1],[9E+09,9E+09,9E+09,9E+09,9E+09,9E+09]];
  CONST robtarget T_815_2:=[[-106.61,355.555,0],[1,0,0,0],[0,0,-1,1],[9E+09,9E+09,9E+09,9E+09,9E+09,9E+09]];
  CONST robtarget T_816_2:=[[-102.152,328.407,0],[1,0,0,0],[0,0,-1,1],[9E+09,9E+09,9E+09,9E+09,9E+09,9E+09]];
  CONST robtarget T_817_2:=[[-119.494,281.892,0],[1,0,0,0],[0,0,-1,1],[9E+09,9E+09,9E+09,9E+09,9E+09,9E+09]];
  CONST robtarget T_818_2:=[[-162.444,263.253,0],[1,0,0,0],[-1,-2,1,1],[9E+09,9E+09,9E+09,9E+09,9E+09,9E+09]];
  CONST robtarget T_819_2:=[[-192.59,272.249,0],[1,0,0,0],[-1,-2,1,1],[9E+09,9E+09,9E+09,9E+09,9E+09,9E+09]];
  CONST robtarget T_820_2:=[[-212.363,298.748,0],[1,0,0,0],[-1,-2,1,1],[9E+09,9E+09,9E+09,9E+09,9E+09,9E+09]];
  CONST robtarget T_821_2:=[[-214.308,359.688,0],[1,0,0,0],[0,1,-2,1],[9E+09,9E+09,9E+09,9E+09,9E+09,9E+09]];
  CONST robtarget T_91_2:=[[-105.556,371.949,0],[1,0,0,0],[0,0,-1,1],[9E+09,9E+09,9E+09,9E+09,9E+09,9E+09]];
  CONST robtarget T_92_2:=[[-102.801,349.258,0],[1,0,0,0],[0,0,-1,1],[9E+09,9E+09,9E+09,9E+09,9E+09,9E+09]];
  CONST robtarget T_93_2:=[[-110.986,309.388,0],[1,0,0,0],[0,0,-1,1],[9E+09,9E+09,9E+09,9E+09,9E+09,9E+09]];
  CONST robtarget T_94_2:=[[-134.729,281.673,0],[1,0,0,0],[-1,-2,1,1],[9E+09,9E+09,9E+09,9E+09,9E+09,9E+09]];
  CONST robtarget T_95_2:=[[-171.682,265.223,0],[1,0,0,0],[-1,-2,1,1],[9E+09,9E+09,9E+09,9E+09,9E+09,9E+09]];
  CONST robtarget T_96_2:=[[-218.684,259.631,0],[1,0,0,0],[-1,-2,1,1],[9E+09,9E+09,9E+09,9E+09,9E+09,9E+09]];
  CONST robtarget T_97_2:=[[-263.903,265.304,0],[1,0,0,0],[-1,-2,1,1],[9E+09,9E+09,9E+09,9E+09,9E+09,9E+09]];
  CONST robtarget T_98_2:=[[-292.752,281.349,0],[1,0,0,0],[-1,-2,1,1],[9E+09,9E+09,9E+09,9E+09,9E+09,9E+09]];
  CONST robtarget T_99_2:=[[-306.123,300.798,0],[1,0,0,0],[-1,-2,1,1],[9E+09,9E+09,9E+09,9E+09,9E+09,9E+09]];
  CONST robtarget T_910_2:=[[-310.742,325.757,0],[1,0,0,0],[-1,-2,1,1],[9E+09,9E+09,9E+09,9E+09,9E+09,9E+09]];
  CONST robtarget T_911_2:=[[-305.799,350.15,0],[1,0,0,0],[0,1,-2,1],[9E+09,9E+09,9E+09,9E+09,9E+09,9E+09]];
  CONST robtarget T_912_2:=[[-291.942,370.49,0],[1,0,0,0],[0,1,-2,1],[9E+09,9E+09,9E+09,9E+09,9E+09,9E+09]];
  CONST robtarget T_913_2:=[[-269.9,384.266,0],[1,0,0,0],[0,1,-2,1],[9E+09,9E+09,9E+09,9E+09,9E+09,9E+09]];
  CONST robtarget T_914_2:=[[-241.699,389.291,0],[1,0,0,0],[0,1,-2,1],[9E+09,9E+09,9E+09,9E+09,9E+09,9E+09]];
  CONST robtarget T_915_2:=[[-211.472,383.78,0],[1,0,0,0],[0,1,-2,1],[9E+09,9E+09,9E+09,9E+09,9E+09,9E+09]];
  CONST robtarget T_916_2:=[[-190.645,367.573,0],[1,0,0,0],[0,1,-2,1],[9E+09,9E+09,9E+09,9E+09,9E+09,9E+09]];
  CONST robtarget T_917_2:=[[-181.245,349.177,0],[1,0,0,0],[-1,-2,1,1],[9E+09,9E+09,9E+09,9E+09,9E+09,9E+09]];
  CONST robtarget T_918_2:=[[-178.814,328.999,0],[1,0,0,0],[-1,-2,1,1],[9E+09,9E+09,9E+09,9E+09,9E+09,9E+09]];
  CONST robtarget T_919_2:=[[-182.136,307.767,0],[1,0,0,0],[-1,-2,1,1],[9E+09,9E+09,9E+09,9E+09,9E+09,9E+09]];
  CONST robtarget T_920_2:=[[-192.752,287.346,0],[1,0,0,0],[-1,-2,1,1],[9E+09,9E+09,9E+09,9E+09,9E+09,9E+09]];
  TASK PERS wobjdata Board:=[FALSE,TRUE,"",[[350,-300,450],[0,0,1,0]],[[0,0,0],[1,0,0,0]]];
ENDMODULE

! task T_ROB1
MODULE MainModule
  VAR robtarget goal:=[[0,0,0],[1,0,0,0],[0,0,0,0],[9E+09,9E+09,9E+09,9E+09,9E+09,9E+09]];
  VAR robtarget targetDraw:=[[0,0,0],[1,0,0,0],[0,0,0,0],[9E+09,9E+09,9E+09,9E+09,9E+09,9E+09]];
  CONST jointtarget jointHome:=[[0,0,0,0,0,0],[0,0,0,0,0,0]];
  PROC connection()
    SetDO DO_01,1;
    SetDO DO_02,0;
    SetDO DO_03,0;
  ENDPROC
  PROC disconnection()
    SetDO DO_01,0;
    SetDO DO_02,1;
    SetDO DO_03,0;
    SetDO DO_04,0;
    SetDO DO_05,1;
  ENDPROC
  PROC getOrders()
    SetDO DO_03,1;
    SetDO DO_04,0;
    SetDO DO_05,1;
    MoveJ goal,generalSpeed,fine,VacuumGripper;
    SetDO DO_05,0;
    SetDO DO_04,1;
    WaitTime 1;
    MoveL Offs(currentPose, 0, 0, -safeHeightObjects),generalSpeed,fine,VacuumGripper;
    WaitTime 1;
    MoveL Offs(currentPose, 0, 0, 100),generalSpeed,fine,VacuumGripper;
    MoveL Offs(currentPose, 0, 0, -safeHeightObjects),generalSpeed,fine,VacuumGripper;
    WaitTime 1;
    SetDO DO_04,0;
    SetDO DO_05,1;
    MoveL Offs(currentPose, 0, 0, 100),generalSpeed,fine,VacuumGripper;
    MoveJ goal,generalSpeed,z10,VacuumGripper;
    MoveL Offs(currentPose, X, Y, Z),generalSpeed,z10,VacuumGripper;
    MoveAbsJ currentJoints,generalSpeed,z10,VacuumGripper;
    MoveJ targetDraw,generalSpeed,z10,VacuumGripper\WObj:=Board;
    MoveJ Offs(currentPose, 0, 0, 100),generalSpeed,z10,VacuumGripper;
    MoveJ targetDraw,generalSpeed,z10,VacuumGripper\WObj:=Board;
    WaitTime 2;
  ENDPROC
  PROC getCommands()
    MoveJ goal,generalSpeed,fine,VacuumGripper;
    MoveL Offs(currentPose, 0, 0, -safeHeightObjects),generalSpeed,fine,VacuumGripper;
    WaitTime 1;
    MoveL Offs(currentPose, 0, 0, 100),generalSpeed,fine,VacuumGripper;
    MoveL Offs(currentPose, 0, 0, -safeHeightObjects),generalSpeed,fine,VacuumGripper;
    WaitTime 1;
    MoveL Offs(currentPose, 0, 0, 100),generalSpeed,fine,VacuumGripper;
    MoveJ goal,generalSpeed,z10,VacuumGripper;
    MoveL Offs(currentPose, X, Y, Z),generalSpeed,z10,VacuumGripper;
    MoveAbsJ currentJoints,generalSpeed,z10,VacuumGripper;
    MoveJ targetDraw,generalSpeed,z10,VacuumGripper\WObj:=Board;
    MoveJ Offs(currentPose, 0, 0, 100),generalSpeed,z10,VacuumGripper;
    MoveJ targetDraw,generalSpeed,z10,VacuumGripper\WObj:=Board;
    WaitTime 2;
  ENDPROC
ENDMODULE

! task T_ROB1
MODULE Parameters
  VAR robtarget currentPose:=[[0,0,0],[1,0,0,0],[0,0,0,0],[9E+09,9E+09,9E+09,9E+09,9E+09,9E+09]];
ENDMODULE


--- Controller Data/IRB140_6_81/RAPID/TASK1/PROGMOD/MainModule.mod ---
MODULE MainModule
    PROC SendMessage(string message)
        ! 0 Scope error to client or end effector error to client | 1 Successful command validation
        SocketSend clientSocket \str := message;
    ENDPROC

    PROC SetGripperState (num state)
        ! DO_03 1 and DO_04 0 -> On | DO_03 0 and DO_04 1 -> Off
        SetDO DO_03, state;
        SetDO DO_04, 1 - state;
    ENDPROC

    PROC PickRoutine(num state)
        SetGripperState(1); ! On vacuum
        MoveL Offs(currentPoint, 0, 0, safeHeightPick), generalSpeed, pickZone, vacuumGripper;
        SetGripperState(state);
        WaitTime(1);
        currentPoint := CRobT(\Tool:=vacuumGripper, \WObj:= wobj0);
        MoveL Offs(currentPoint, 0, 0, heightObjects), generalSpeed, pickZone, vacuumGripper;
        SendMessage("1");
    ENDPROC

    PROC PickCommand()
        IF commandValue = 2 THEN ! Absolute drop
            SetGripperState(0); ! Off vacuum
            SendMessage("1");
        ELSE
            IF goalPoint.trans.z < safeZ THEN
                SendMessage("0");
            ELSE
                MoveJ goalPoint, generalSpeed, pickZone, vacuumGripper;
                currentPoint := CRobT(\Tool:=vacuumGripper, \WObj:= wobj0);
                IF commandValue = 1 THEN ! Pick object
                    PickRoutine(1);
                ELSE ! Drop object
                    PickRoutine(0);
                ENDIF
            ENDIF
        ENDIF
    ENDPROC

    PROC String2CommandParameters(string stringData)
        VAR num lengthString;
        VAR num initialIndex := 1;
        VAR num indexArray;
        VAR string strVals {9};
        VAR bool parsedOk {9};
        FOR i FROM 0 TO 8 DO
            indexArray := i + 1;
            lengthString := lengthStrings{indexArray};
            strVals{indexArray} := StrPart(stringData, initialIndex, lengthString);
            initialIndex := initialIndex + lengthString;
        ENDFOR
        parsedOk := [StrToVal(strVals{1}, x), StrToVal(strVals{2}, y), StrToVal(strVals{3}, z),
                     StrToVal(strVals{4}, qw), StrToVal(strVals{5}, q1), StrToVal(strVals{6}, q2),
                     StrToVal(strVals{7}, q3), StrToVal(strVals{8}, command), StrToVal(strVals{9}, commandValue)];
    ENDPROC

    FUNC bool NotReachable(robtarget pointToReach, PERS tooldata tool, PERS wobjdata workObject)
        VAR jointtarget jointsCalculation;
        VAR bool notReachable := FALSE;
        jointsCalculation := CalcJointT(pointToReach, tool \Wobj := workObject);
        RETURN notReachable;
        ERROR
        IF ERRNO = ERR_ROBLIMIT OR ERRNO = ERR_OUTSIDE_REACH THEN
            notReachable := TRUE;
            TRYNEXT;
        ENDIF
    ENDFUNC

    PROC MoveCommand()
        VAR num futureZ;
        IF commandValue = 0 THEN ! MoveJ
            IF NotReachable(goalPoint, vacuumGripper, wobj0) OR goalPoint.trans.z < safeZ THEN
                SendMessage("0");
            ELSE
                MoveJ goalPoint, generalSpeed, generalZone, vacuumGripper;
                SendMessage("1");
            ENDIF
        ELSE !MoveL
            currentPoint := CRobT(\Tool:=vacuumGripper, \WObj:= wobj0);
            futureZ := currentPoint.trans.z + z;
            IF futureZ < safeZ THEN
                SendMessage("0");
            ELSE
                MoveL Offs(currentPoint, x, y, z), generalSpeed, generalZone, vacuumGripper;
                SendMessage("1");
            ENDIF
        ENDIF
        ERROR
    ENDPROC

    PROC RotateCommand()
        VAR jointtarget currentJoints;
        VAR jointtarget futureJoints;
        currentJoints := CJointT();
        futureJoints := currentJoints;
        futureJoints.robax.rax_6 := futureJoints.robax.rax_6 + commandValue;
        MoveAbsJ futureJoints, generalSpeed, generalZone, vacuumGripper;
        SendMessage("1");
    ENDPROC

    FUNC bool DrawNumber(num digit, num offset)
        VAR num indexPointNumber;
        VAR robtarget numberPoint;
        FOR i FROM 0 TO amountPoints{digit + 1} DO
            indexPointNumber := startIndices{digit + 1} + i;
            numberPoint := numbersPoints{indexPointNumber};
            numberPoint.trans.y := numberPoint.trans.y + offset;
            MoveJ numberPoint, generalSpeed, generalZone, vacuumGripper \WObj := drawBoard;
        ENDFOR
        RETURN TRUE;
    ENDFUNC

    PROC DrawCommand()
        VAR num tens;
        VAR num units;
        VAR bool digitDrawn;
        units := commandValue;
        IF commandValue > 9 THEN
            tens := Trunc(commandValue / 10);
            units := commandValue - tens * 10;
            digitDrawn := DrawNumber(tens, tensOffset);
            currentPoint := CRobT(\Tool :=vacuumGripper, \WObj := wobj0);
            MoveJ Offs(currentPoint, 0, 0, 100), generalSpeed, generalZone, vacuumGripper;
        ENDIF
        digitDrawn := DrawNumber(units, -tensOffset);
        SendMessage("1");
    ENDPROC

    PROC GetCommand()
        VAR string clientData;
        SocketReceive clientSocket \str := clientData \Time:= WAIT_MAX; ! Data from client
        String2CommandParameters(clientData); ! String data to numbers
        goalPoint := [[x, y, z],[qw, q1, q2, q3],[0, 0, 0, 0],[9E9, 9E9, 9E9, 9E9, 9E9, 9E9]]; ! Create goalPoint robTarget
        IF command = 0 THEN ! Pick
            PickCommand;
        ELSEIF command = 1 THEN ! Move
            MoveCommand;
        ELSEIF command = 2 THEN ! Rotate
            RotateCommand;
        ELSEIF command = 3 THEN ! Draw
            DrawCommand;
        ENDIF
        WaitTime(2); ! Before the next command
    ENDPROC

    PROC GoHome()
        MoveAbsJ homeJoints, generalSpeed, generalZone, tool0;
    ENDPROC

    PROC SocketDisconnection()
        SocketClose clientSocket;
        SocketClose serverSocket;
        clientConnected := FALSE;
        SetDO DO_01, 0; ! Off lamp 1 -> It is not connected
        SetDO DO_02, 1; ! On lamp 2 -> It is disconnected
        SetGripperState(0); ! Off vacuum
        GoHome;
    ENDPROC

    PROC SocketConnection()
        SocketCreate serverSocket;
        SocketBind serverSocket, ipController, 8000;
        SocketListen serverSocket;
        SocketAccept serverSocket, clientSocket, \Time := WAIT_MAX ;
        clientConnected := TRUE;
        SocketSend clientSocket \str := "Success";
        SetDO DO_01, 1; ! On lamp 1 -> It is connected
        SetDO DO_02, 0; ! Off lamp 2 -> It is not disconnected
    ENDPROC

    PROC main()
        SocketDisconnection;
        WHILE TRUE DO
            IF (NOT clientConnected) AND DI_01 = 1 THEN ! Connection
                SocketConnection;
            ELSEIF DI_02 = 1 THEN ! Disconnection
                SocketDisconnection;
            ELSEIF clientConnected THEN ! Getting commands
                GetCommand;
            ENDIF
        ENDWHILE
    ENDPROC
ENDMODULE

--- Controller Data/IRB140_6_81/RAPID/TASK1/PROGMOD/Numbers.mod ---
MODULE Numbers
    ! Zero points
    CONST robtarget P_01 := [[-310.742,318.894,0],[1,0,0,0],[0,0,0,0],[9E+09,9E+09,9E+09,9E+09,9E+09,9E+09]];
    CONST robtarget P_02 := [[-285.702,367.273,0],[1,0,0,0],[0,0,0,0],[9E+09,9E+09,9E+09,9E+09,9E+09,9E+09]];
    CONST robtarget P_03 := [[-206.529,382.913,0],[1,0,0,0],[0,0,0,0],[9E+09,9E+09,9E+09,9E+09,9E+09,9E+09]];
    CONST robtarget P_04 := [[-128.165,367.435,0],[1,0,0,0],[0,0,0,0],[9E+09,9E+09,9E+09,9E+09,9E+09,9E+09]];
    CONST robtarget P_05 := [[-102.477,318.894,0],[1,0,0,0],[0,0,0,0],[9E+09,9E+09,9E+09,9E+09,9E+09,9E+09]];
    CONST robtarget P_06 := [[-127.679,270.676,0],[1,0,0,0],[0,0,0,0],[9E+09,9E+09,9E+09,9E+09,9E+09,9E+09]];
    CONST robtarget P_07 := [[-206.691,255.036,0],[1,0,0,0],[0,0,0,0],[9E+09,9E+09,9E+09,9E+09,9E+09,9E+09]];
    CONST robtarget P_08 := [[-284.811,270.514,0],[1,0,0,0],[0,0,0,0],[9E+09,9E+09,9E+09,9E+09,9E+09,9E+09]];
    CONST robtarget P_09 := [[-310.742,318.894,0],[1,0,0,0],[0,0,0,0],[9E+09,9E+09,9E+09,9E+09,9E+09,9E+09]];
    ! One points
    CONST robtarget P_11 := [[-106.691,366.707,0],[1,0,0,0],[0,0,0,0],[9E+09,9E+09,9E+09,9E+09,9E+09,9E+09]];
    CONST robtarget P_12 := [[-106.691,269.138,0],[1,0,0,0],[0,0,0,0],[9E+09,9E+09,9E+09,9E+09,9E+09,9E+09]];
    CONST robtarget P_13 := [[-106.691,317.923,0],[1,0,0,0],[0,0,0,0],[9E+09,9E+09,9E+09,9E+09,9E+09,9E+09]];
    CONST robtarget P_14 := [[-307.339,315.005,0],[1,0,0,0],[0,0,0,0],[9E+09,9E+09,9E+09,9E+09,9E+09,9E+09]];
    CONST robtarget P_15 := [[-285.297,336.399,0],[1,0,0,0],[0,0,0,0],[9E+09,9E+09,9E+09,9E+09,9E+09,9E+09]];
    CONST robtarget P_16 := [[-279.462,366.707,0],[1,0,0,0],[0,0,0,0],[9E+09,9E+09,9E+09,9E+09,9E+09,9E+09]];
    ! Two points
    CONST robtarget P_21 := [[-106.691,261.009,0],[1,0,0,0],[0,0,0,0],[9E+09,9E+09,9E+09,9E+09,9E+09,9E+09]];
    CONST robtarget P_22 := [[-106.691,384.347,0],[1,0,0,0],[0,0,0,0],[9E+09,9E+09,9E+09,9E+09,9E+09,9E+09]];
    CONST robtarget P_23 := [[-129.867,359.226,0],[1,0,0,0],[0,0,0,0],[9E+09,9E+09,9E+09,9E+09,9E+09,9E+09]];
    CONST robtarget P_24 := [[-153.206,334.509,0],[1,0,0,0],[0,0,0,0],[9E+09,9E+09,9E+09,9E+09,9E+09,9E+09]];
    CONST robtarget P_25 := [[-181.731,306.39,0],[1,0,0,0],[0,0,0,0],[9E+09,9E+09,9E+09,9E+09,9E+09,9E+09]];
    CONST robtarget P_26 := [[-215.929,279.647,0],[1,0,0,0],[0,0,0,0],[9E+09,9E+09,9E+09,9E+09,9E+09,9E+09]];
    CONST robtarget P_27 := [[-255.961,269.274,0],[1,0,0,0],[0,0,0,0],[9E+09,9E+09,9E+09,9E+09,9E+09,9E+09]];
    CONST robtarget P_28 := [[-296.075,285.077,0],[1,0,0,0],[0,0,0,0],[9E+09,9E+09,9E+09,9E+09,9E+09,9E+09]];
    CONST robtarget P_29 := [[-310.905,328.918,0],[1,0,0,0],[0,0,0,0],[9E+09,9E+09,9E+09,9E+09,9E+09,9E+09]];
    CONST robtarget P_210 := [[-306.934,357.038,0],[1,0,0,0],[0,0,0,0],[9E+09,9E+09,9E+09,9E+09,9E+09,9E+09]];
    CONST robtarget P_211 := [[-298.911,380.133,0],[1,0,0,0],[0,0,0,0],[9E+09,9E+09,9E+09,9E+09,9E+09,9E+09]];
    ! Three points
    CONST robtarget P_31 := [[-298.587,375.377,0],[1,0,0,0],[0,0,0,0],[9E+09,9E+09,9E+09,9E+09,9E+09,9E+09]];
    CONST robtarget P_32 := [[-307.096,351.633,0],[1,0,0,0],[0,0,0,0],[9E+09,9E+09,9E+09,9E+09,9E+09,9E+09]];
    CONST robtarget P_33 := [[-310.905,323.189,0],[1,0,0,0],[0,0,0,0],[9E+09,9E+09,9E+09,9E+09,9E+09,9E+09]];
    CONST robtarget P_34 := [[-308.149,299.445,0],[1,0,0,0],[0,0,0,0],[9E+09,9E+09,9E+09,9E+09,9E+09,9E+09]];
    CONST robtarget P_35 := [[-299.559,281.049,0],[1,0,0,0],[0,0,0,0],[9E+09,9E+09,9E+09,9E+09,9E+09,9E+09]];
    CONST robtarget P_36 := [[-284.081,267.759,0],[1,0,0,0],[0,0,0,0],[9E+09,9E+09,9E+09,9E+09,9E+09,9E+09]];
    CONST robtarget P_37 := [[-262.606,263.221,0],[1,0,0,0],[0,0,0,0],[9E+09,9E+09,9E+09,9E+09,9E+09,9E+09]];
    CONST robtarget P_38 := [[-233.595,274.08,0],[1,0,0,0],[0,0,0,0],[9E+09,9E+09,9E+09,9E+09,9E+09,9E+09]];
    CONST robtarget P_39 := [[-217.874,300.174,0],[1,0,0,0],[0,0,0,0],[9E+09,9E+09,9E+09,9E+09,9E+09,9E+09]];
    CONST robtarget P_310 := [[-215.199,340.044,0],[1,0,0,0],[0,0,0,0],[9E+09,9E+09,9E+09,9E+09,9E+09,9E+09]];
    CONST robtarget P_311 := [[-215.929,300.174,0],[1,0,0,0],[0,0,0,0],[9E+09,9E+09,9E+09,9E+09,9E+09,9E+09]];
    CONST robtarget P_312 := [[-202.963,273.27,0],[1,0,0,0],[0,0,0,0],[9E+09,9E+09,9E+09,9E+09,9E+09,9E+09]];
    CONST robtarget P_313 := [[-188.214,263.221,0],[1,0,0,0],[0,0,0,0],[9E+09,9E+09,9E+09,9E+09,9E+09,9E+09]];
    CONST robtarget P_314 := [[-166.01,259.331,0],[1,0,0,0],[0,0,0,0],[9E+09,9E+09,9E+09,9E+09,9E+09,9E+09]];
    CONST robtarget P_315 := [[-141.131,263.95,0],[1,0,0,0],[0,0,0,0],[9E+09,9E+09,9E+09,9E+09,9E+09,9E+09]];
    CONST robtarget P_316 := [[-120.953,276.997,0],[1,0,0,0],[0,0,0,0],[9E+09,9E+09,9E+09,9E+09,9E+09,9E+09]];
    CONST robtarget P_317 := [[-107.177,298.148,0],[1,0,0,0],[0,0,0,0],[9E+09,9E+09,9E+09,9E+09,9E+09,9E+09]];
    CONST robtarget P_318 := [[-102.477,326.268,0],[1,0,0,0],[0,0,0,0],[9E+09,9E+09,9E+09,9E+09,9E+09,9E+09]];
    CONST robtarget P_319 := [[-106.123,356.09,0],[1,0,0,0],[0,0,0,0],[9E+09,9E+09,9E+09,9E+09,9E+09,9E+09]];
    CONST robtarget P_320 := [[-114.794,380.887,0],[1,0,0,0],[0,0,0,0],[9E+09,9E+09,9E+09,9E+09,9E+09,9E+09]];
    ! Four points
    CONST robtarget P_41 := [[-106.691,281.323,0],[1,0,0,0],[0,0,0,0],[9E+09,9E+09,9E+09,9E+09,9E+09,9E+09]];
    CONST robtarget P_42 := [[-306.691,281.323,0],[1,0,0,0],[0,0,0,0],[9E+09,9E+09,9E+09,9E+09,9E+09,9E+09]];
    CONST robtarget P_43 := [[-306.691,305.958,0],[1,0,0,0],[0,0,0,0],[9E+09,9E+09,9E+09,9E+09,9E+09,9E+09]];
    CONST robtarget P_44 := [[-203.611,395.424,0],[1,0,0,0],[0,0,0,0],[9E+09,9E+09,9E+09,9E+09,9E+09,9E+09]];
    CONST robtarget P_45 := [[-175.41,395.424,0],[1,0,0,0],[0,0,0,0],[9E+09,9E+09,9E+09,9E+09,9E+09,9E+09]];
    CONST robtarget P_46 := [[-175.41,257.498,0],[1,0,0,0],[0,0,0,0],[9E+09,9E+09,9E+09,9E+09,9E+09,9E+09]];
    ! Five points
    CONST robtarget P_51 := [[-306.691,269.007,0],[1,0,0,0],[0,0,0,0],[9E+09,9E+09,9E+09,9E+09,9E+09,9E+09]];
    CONST robtarget P_52 := [[-306.691,378.732,0],[1,0,0,0],[0,0,0,0],[9E+09,9E+09,9E+09,9E+09,9E+09,9E+09]];
    CONST robtarget P_53 := [[-223.611,378.732,0],[1,0,0,0],[0,0,0,0],[9E+09,9E+09,9E+09,9E+09,9E+09,9E+09]];
    CONST robtarget P_54 := [[-229.867,352.962,0],[1,0,0,0],[0,0,0,0],[9E+09,9E+09,9E+09,9E+09,9E+09,9E+09]];
    CONST robtarget P_55 := [[-231.002,334.809,0],[1,0,0,0],[0,0,0,0],[9E+09,9E+09,9E+09,9E+09,9E+09,9E+09]];
    CONST robtarget P_56 := [[-228.49,308.796,0],[1,0,0,0],[0,0,0,0],[9E+09,9E+09,9E+09,9E+09,9E+09,9E+09]];
    CONST robtarget P_57 := [[-218.522,288.456,0],[1,0,0,0],[0,0,0,0],[9E+09,9E+09,9E+09,9E+09,9E+09,9E+09]];
    CONST robtarget P_58 := [[-199.721,273.221,0],[1,0,0,0],[0,0,0,0],[9E+09,9E+09,9E+09,9E+09,9E+09,9E+09]];
    CONST robtarget P_59 := [[-170.224,267.873,0],[1,0,0,0],[0,0,0,0],[9E+09,9E+09,9E+09,9E+09,9E+09,9E+09]];
    CONST robtarget P_510 := [[-143.482,272.492,0],[1,0,0,0],[0,0,0,0],[9E+09,9E+09,9E+09,9E+09,9E+09,9E+09]];
    CONST robtarget P_511 := [[-122.088,285.539,0],[1,0,0,0],[0,0,0,0],[9E+09,9E+09,9E+09,9E+09,9E+09,9E+09]];
    CONST robtarget P_512 := [[-107.744,306.527,0],[1,0,0,0],[0,0,0,0],[9E+09,9E+09,9E+09,9E+09,9E+09,9E+09]];
    CONST robtarget P_513 := [[-102.477,334.647,0],[1,0,0,0],[0,0,0,0],[9E+09,9E+09,9E+09,9E+09,9E+09,9E+09]];
    CONST robtarget P_514 := [[-105.637,362.848,0],[1,0,0,0],[0,0,0,0],[9E+09,9E+09,9E+09,9E+09,9E+09,9E+09]];
    CONST robtarget P_515 := [[-113.822,386.997,0],[1,0,0,0],[0,0,0,0],[9E+09,9E+09,9E+09,9E+09,9E+09,9E+09]];
    ! Six points
    CONST robtarget P_61 := [[-307.663,280.947,0],[1,0,0,0],[0,0,0,0],[9E+09,9E+09,9E+09,9E+09,9E+09,9E+09]];
    CONST robtarget P_62 := [[-310.418,303.638,0],[1,0,0,0],[0,0,0,0],[9E+09,9E+09,9E+09,9E+09,9E+09,9E+09]];
    CONST robtarget P_63 := [[-301.909,343.346,0],[1,0,0,0],[0,0,0,0],[9E+09,9E+09,9E+09,9E+09,9E+09,9E+09]];
    CONST robtarget P_64 := [[-278.165,371.385,0],[1,0,0,0],[0,0,0,0],[9E+09,9E+09,9E+09,9E+09,9E+09,9E+09]];
    CONST robtarget P_65 := [[-241.618,387.916,0],[1,0,0,0],[0,0,0,0],[9E+09,9E+09,9E+09,9E+09,9E+09,9E+09]];
    CONST robtarget P_66 := [[-194.535,393.265,0],[1,0,0,0],[0,0,0,0],[9E+09,9E+09,9E+09,9E+09,9E+09,9E+09]];
    CONST robtarget P_67 := [[-149.721,387.43,0],[1,0,0,0],[0,0,0,0],[9E+09,9E+09,9E+09,9E+09,9E+09,9E+09]];
    CONST robtarget P_68 := [[-120.629,371.223,0],[1,0,0,0],[0,0,0,0],[9E+09,9E+09,9E+09,9E+09,9E+09,9E+09]];
    CONST robtarget P_69 := [[-107.015,351.693,0],[1,0,0,0],[0,0,0,0],[9E+09,9E+09,9E+09,9E+09,9E+09,9E+09]];
    CONST robtarget P_610 := [[-102.477,327.138,0],[1,0,0,0],[0,0,0,0],[9E+09,9E+09,9E+09,9E+09,9E+09,9E+09]];
    CONST robtarget P_611 := [[-107.258,302.503,0],[1,0,0,0],[0,0,0,0],[9E+09,9E+09,9E+09,9E+09,9E+09,9E+09]];
    CONST robtarget P_612 := [[-121.277,282.406,0],[1,0,0,0],[0,0,0,0],[9E+09,9E+09,9E+09,9E+09,9E+09,9E+09]];
    CONST robtarget P_613 := [[-143.076,268.71,0],[1,0,0,0],[0,0,0,0],[9E+09,9E+09,9E+09,9E+09,9E+09,9E+09]];
    CONST robtarget P_614 := [[-171.52,263.605,0],[1,0,0,0],[0,0,0,0],[9E+09,9E+09,9E+09,9E+09,9E+09,9E+09]];
    CONST robtarget P_615 := [[-201.504,268.954,0],[1,0,0,0],[0,0,0,0],[9E+09,9E+09,9E+09,9E+09,9E+09,9E+09]];
    CONST robtarget P_616 := [[-222.574,285.323,0],[1,0,0,0],[0,0,0,0],[9E+09,9E+09,9E+09,9E+09,9E+09,9E+09]];
    CONST robtarget P_617 := [[-232.055,303.638,0],[1,0,0,0],[0,0,0,0],[9E+09,9E+09,9E+09,9E+09,9E+09,9E+09]];
    CONST robtarget P_618 := [[-234.405,324.059,0],[1,0,0,0],[0,0,0,0],[9E+09,9E+09,9E+09,9E+09,9E+09,9E+09]];
    CONST robtarget P_619 := [[-230.759,346.101,0],[1,0,0,0],[0,0,0,0],[9E+09,9E+09,9E+09,9E+09,9E+09,9E+09]];
    CONST robtarget P_620 := [[-220.467,365.712,0],[1,0,0,0],[0,0,0,0],[9E+09,9E+09,9E+09,9E+09,9E+09,9E+09]];
    CONST robtarget P_621 := [[-194.535,393.265,0],[1,0,0,0],[0,0,0,0],[9E+09,9E+09,9E+09,9E+09,9E+09,9E+09]];
    ! Seven points
    CONST robtarget P_71 := [[-306.691,388.239,0],[1,0,0,0],[0,0,0,0],[9E+09,9E+09,9E+09,9E+09,9E+09,9E+09]];
    CONST robtarget P_72 := [[-306.691,261.334,0],[1,0,0,0],[0,0,0,0],[9E+09,9E+09,9E+09,9E+09,9E+09,9E+09]];
    CONST robtarget P_73 := [[-106.691,347.882,0],[1,0,0,0],[0,0,0,0],[9E+09,9E+09,9E+09,9E+09,9E+09,9E+09]];
    ! Eight points
    CONST robtarget P_81 := [[-214.308,359.688,0],[1,0,0,0],[0,0,0,0],[9E+09,9E+09,9E+09,9E+09,9E+09,9E+09]];
    CONST robtarget P_82 := [[-233.109,381.568,0],[1,0,0,0],[-1,0,-1,0],[9E+09,9E+09,9E+09,9E+09,9E+09,9E+09]];
    CONST robtarget P_83 := [[-258.554,388.699,0],[1,0,0,0],[-1,0,-1,0],[9E+09,9E+09,9E+09,9E+09,9E+09,9E+09]];
    CONST robtarget P_84 := [[-296.156,371.681,0],[1,0,0,0],[-1,0,-1,0],[9E+09,9E+09,9E+09,9E+09,9E+09,9E+09]];
    CONST robtarget P_85 := [[-311.229,328.407,0],[1,0,0,0],[-1,0,-1,0],[9E+09,9E+09,9E+09,9E+09,9E+09,9E+09]];
    CONST robtarget P_86 := [[-296.966,284.728,0],[1,0,0,0],[-1,0,-1,0],[9E+09,9E+09,9E+09,9E+09,9E+09,9E+09]];
    CONST robtarget P_87 := [[-260.337,268.278,0],[1,0,0,0],[-1,0,-1,0],[9E+09,9E+09,9E+09,9E+09,9E+09,9E+09]];
    CONST robtarget P_88 := [[-233.757,276.138,0],[1,0,0,0],[-1,0,-1,0],[9E+09,9E+09,9E+09,9E+09,9E+09,9E+09]];
    CONST robtarget P_89 := [[-213.174,298.748,0],[1,0,0,0],[-1,0,-1,0],[9E+09,9E+09,9E+09,9E+09,9E+09,9E+09]];
    CONST robtarget P_810 := [[-213.498,359.688,0],[1,0,0,0],[-1,0,-1,0],[9E+09,9E+09,9E+09,9E+09,9E+09,9E+09]];
    CONST robtarget P_811 := [[-191.78,384.89,0],[1,0,0,0],[-1,0,-1,0],[9E+09,9E+09,9E+09,9E+09,9E+09,9E+09]];
    CONST robtarget P_812 := [[-161.958,393.561,0],[1,0,0,0],[-1,0,-1,0],[9E+09,9E+09,9E+09,9E+09,9E+09,9E+09]];
    CONST robtarget P_813 := [[-138.457,389.185,0],[1,0,0,0],[-1,0,-1,0],[9E+09,9E+09,9E+09,9E+09,9E+09,9E+09]];
    CONST robtarget P_814 := [[-119.332,376.381,0],[1,0,0,0],[-1,0,-1,0],[9E+09,9E+09,9E+09,9E+09,9E+09,9E+09]];
    CONST robtarget P_815 := [[-106.61,355.555,0],[1,0,0,0],[-1,0,-1,0],[9E+09,9E+09,9E+09,9E+09,9E+09,9E+09]];
    CONST robtarget P_816 := [[-102.152,328.407,0],[1,0,0,0],[-1,0,-1,0],[9E+09,9E+09,9E+09,9E+09,9E+09,9E+09]];
    CONST robtarget P_817 := [[-119.494,281.892,0],[1,0,0,0],[0,0,0,0],[9E+09,9E+09,9E+09,9E+09,9E+09,9E+09]];
    CONST robtarget P_818 := [[-162.444,263.253,0],[1,0,0,0],[0,0,0,0],[9E+09,9E+09,9E+09,9E+09,9E+09,9E+09]];
    CONST robtarget P_819 := [[-192.59,272.249,0],[1,0,0,0],[0,0,0,0],[9E+09,9E+09,9E+09,9E+09,9E+09,9E+09]];
    CONST robtarget P_820 := [[-212.363,298.748,0],[1,0,0,0],[0,0,0,0],[9E+09,9E+09,9E+09,9E+09,9E+09,9E+09]];
    CONST robtarget P_821 := [[-214.308,359.688,0],[1,0,0,0],[0,0,0,0],[9E+09,9E+09,9E+09,9E+09,9E+09,9E+09]];
    ! Nine points
    CONST robtarget P_91 := [[-105.556,371.949,0],[1,0,0,0],[0,0,0,0],[9E+09,9E+09,9E+09,9E+09,9E+09,9E+09]];
    CONST robtarget P_92 := [[-102.801,349.258,0],[1,0,0,0],[-1,0,-1,0],[9E+09,9E+09,9E+09,9E+09,9E+09,9E+09]];
    CONST robtarget P_93 := [[-110.986,309.388,0],[1,0,0,0],[-1,0,-1,0],[9E+09,9E+09,9E+09,9E+09,9E+09,9E+09]];
    CONST robtarget P_94 := [[-134.729,281.673,0],[1,0,0,0],[-1,0,-1,0],[9E+09,9E+09,9E+09,9E+09,9E+09,9E+09]];
    CONST robtarget P_95 := [[-171.682,265.223,0],[1,0,0,0],[-1,0,-1,0],[9E+09,9E+09,9E+09,9E+09,9E+09,9E+09]];
    CONST robtarget P_96 := [[-218.684,259.631,0],[1,0,0,0],[-1,0,-1,0],[9E+09,9E+09,9E+09,9E+09,9E+09,9E+09]];
    CONST robtarget P_97 := [[-263.903,265.304,0],[1,0,0,0],[-1,0,-1,0],[9E+09,9E+09,9E+09,9E+09,9E+09,9E+09]];
    CONST robtarget P_98 := [[-292.752,281.349,0],[1,0,0,0],[0,0,0,0],[9E+09,9E+09,9E+09,9E+09,9E+09,9E+09]];
    CONST robtarget P_99 := [[-306.123,300.798,0],[1,0,0,0],[0,0,0,0],[9E+09,9E+09,9E+09,9E+09,9E+09,9E+09]];
    CONST robtarget P_910 := [[-310.742,325.757,0],[1,0,0,0],[0,0,0,0],[9E+09,9E+09,9E+09,9E+09,9E+09,9E+09]];
    CONST robtarget P_911 := [[-305.799,350.15,0],[1,0,0,0],[0,0,0,0],[9E+09,9E+09,9E+09,9E+09,9E+09,9E+09]];
    CONST robtarget P_912 := [[-291.942,370.49,0],[1,0,0,0],[0,0,0,0],[9E+09,9E+09,9E+09,9E+09,9E+09,9E+09]];
    CONST robtarget P_913 := [[-269.9,384.266,0],[1,0,0,0],[0,0,0,0],[9E+09,9E+09,9E+09,9E+09,9E+09,9E+09]];
    CONST robtarget P_914 := [[-241.699,389.291,0],[1,0,0,0],[0,0,0,0],[9E+09,9E+09,9E+09,9E+09,9E+09,9E+09]];
    CONST robtarget P_915 := [[-211.472,383.78,0],[1,0,0,0],[0,0,0,0],[9E+09,9E+09,9E+09,9E+09,9E+09,9E+09]];
    CONST robtarget P_916 := [[-190.645,367.573,0],[1,0,0,0],[0,0,0,0],[9E+09,9E+09,9E+09,9E+09,9E+09,9E+09]];
    CONST robtarget P_917 := [[-181.245,349.177,0],[1,0,0,0],[0,0,0,0],[9E+09,9E+09,9E+09,9E+09,9E+09,9E+09]];
    CONST robtarget P_918 := [[-178.814,328.999,0],[1,0,0,0],[0,0,0,0],[9E+09,9E+09,9E+09,9E+09,9E+09,9E+09]];
    CONST robtarget P_919 := [[-182.136,307.767,0],[1,0,0,0],[0,0,0,0],[9E+09,9E+09,9E+09,9E+09,9E+09,9E+09]];
    CONST robtarget P_920 := [[-192.752,287.346,0],[1,0,0,0],[0,0,0,0],[9E+09,9E+09,9E+09,9E+09,9E+09,9E+09]];
    CONST robtarget P_921 := [[-218.684,259.631,0],[1,0,0,0],[0,0,0,0],[9E+09,9E+09,9E+09,9E+09,9E+09,9E+09]];
    ! Numbers array
    CONST robtarget numbersPoints{133} := [P_01, P_02, P_03, P_04, P_05, P_06, P_07, P_08, P_09,
                                           P_11, P_12, P_13, P_14, P_15, P_16, P_21, P_22, P_23,
                                           P_24, P_25, P_26, P_27, P_28, P_29, P_210, P_211, P_31,
                                           P_32, P_33, P_34, P_35, P_36, P_37, P_38, P_39, P_310,
                                           P_311, P_312, P_313, P_314, P_315, P_316, P_317, P_318,
                                           P_319, P_320, P_41, P_42, P_43, P_44, P_45, P_46, P_51,
                                           P_52, P_53, P_54, P_55, P_56, P_57, P_58, P_59, P_510,
                                           P_511, P_512, P_513, P_514, P_515, P_61, P_62, P_63,
                                           P_64, P_65, P_66, P_67, P_68, P_69, P_610, P_611, P_612,
                                           P_613, P_614, P_615, P_616, P_617, P_618, P_619, P_620,
                                           P_621, P_71, P_72, P_73, P_81, P_82, P_83, P_84, P_85,
                                           P_86, P_87, P_88, P_89, P_810, P_811, P_812, P_813, P_814,
                                           P_815, P_816, P_817, P_818, P_819, P_820, P_821, P_91, P_92,
                                           P_93, P_94, P_95, P_96, P_97, P_98, P_99, P_910, P_911, P_912,
                                           P_913, P_914, P_915, P_916, P_917, P_918,P_919, P_920, P_921];
    CONST num amountPoints{10} := [8, 5, 10, 19, 5, 14, 20, 2, 20, 20]; ! Amount of points per number
    CONST num startIndices{10} := [1, 10, 16, 27, 47, 53, 68, 89, 92, 113];
ENDMODULE

--- Controller Data/IRB140_6_81/RAPID/TASK1/PROGMOD/Parameters.mod ---
MODULE Parameters
    ! Socket global parameters
    ! Simulated controller ip "127.0.0.1" | Real robot controller ip "192.168.125.1"
    CONST string ipController := "127.0.0.1";
    VAR socketdev serverSocket;
    VAR socketdev clientSocket;
    VAR bool clientConnected;
    VAR num x;
    VAR num y;
    VAR num z;
    VAR num qw;
    VAR num q1;
    VAR num q2;
    VAR num q3;
    VAR num command;
    VAR num commandValue;
    VAR robtarget goalPoint;
    ! Safety parameters
    CONST num safeZ := 150;
    CONST num heightObjects := 100;
    ! For real environment the offsetHeightPick is 5
    CONST num offsetHeightPick := 0;
    CONST num safeHeightPick := offsetHeightPick - heightObjects;
    ! Controller parameters
    CONST num lengthStrings {9} := [4, 4, 4, 12, 12, 12, 12, 1, 4];
    CONST num tensOffset := 70;
    CONST speeddata generalSpeed := v80;
    CONST zonedata generalZone := z10;
    CONST zonedata pickZone := fine;
    CONST jointtarget homeJoints := [[0, 0, 0, 0, 0, 0],[0, 0, 0, 0, 0, 0]];
    PERS tooldata vacuumGripper := [TRUE, [[0, 0, 129.78],[1, 0, 0, 0]],[1, [0, 0, 1],[1, 0, 0, 0], 0, 0, 0]];
    PERS wobjdata drawBoard := [FALSE,TRUE,"",[[350,-300,450],[0,0,1,0]],[[0,0,0],[1,0,0,0]]];
    VAR robtarget currentPoint;
ENDMODULE

--- Controller Data/IRB140_6_81/SYSPAR/EIO.cfg ---
EIO:CFG_1.0:6:1::
#
EIO_SIGNAL:

      -Name "DI_01" -SignalType "DI"

      -Name "DI_02" -SignalType "DI"

      -Name "DO_01" -SignalType "DO"

      -Name "DO_02" -SignalType "DO"

      -Name "DO_03" -SignalType "DO"

      -Name "DO_04" -SignalType "DO"
